// TIA Portal V19 export
TYPE "LEXCHANGETRAY_typeVfd_cmd"
// stored: Access Published
   STRUCT
      simActive : Bool;   // Simulation Mode Active Flag
      enable : Bool;   // VFD Enable Command
      reset : Bool;   // VFD Reset Command
      enableManualCmds : Bool;   // Enable Manual Control Mode
      interlock : Bool;   // Safety Interlock Signal
      downloadRampTime : Bool;   // Download Acceleration/Deceleration Ramp Times
      statVfdSportsIncEnable : Bool;   // VFD Sports Mode Increment Enable Status
      statVfdSportsIncReset : Bool;   // VFD Sports Mode Increment Reset Status
   END_STRUCT;
END_TYPE
